{attribute 'qualified_only'}
{attribute 'strict'}
TYPE E_StateDescription :
(
	Undefined		:= 0,
	Off				:= 10,
	SelfTest		:= 20,
	Maintenance 	:= 30,
	OutOfService 	:= 40,
	Idle			:= 50,
	ServingCustomer	:= 60
);
END_TYPE

(* stored: Version 1.1.0.1, ProductVersion 3.1.4024.12
   DUT E_StateDescription: Id {c7a59eda-44d9-04ee-31d3-5db7bf9ca168} *)
